{attribute 'enable_dynamic_creation'}
TYPE ST_LoggerNode :
STRUCT
	iLogger:			I_Logger;
	pNext: 				POINTER TO ST_LoggerNode;
END_STRUCT
END_TYPE

(* stored: Version 1.1.0.1
   DUT ST_LoggerNode: Id {b56b6f89-5e19-42c9-aa25-77242f785d37} *)
